{library PUBLIC}
(* Station number type *)
TYPE StationType : INT(1..9);
END_TYPE

(* stored: Version 1.1.0.1, ProductVersion 3.1.4022.12
   EnumerationTextList StationType: Id {84364646-8757-4457-9d8c-def0b77cb768} *)
